PROGRAM P_IncAusstossV
VAR
END_VAR

IF DB6.rAusstossverz < 0.91 THEN
	DB6.rAusstossverz := DB6.rAusstossverz + 0.1;
	DB6.nAusstossverz := REAL_TO_INT(DB6.rAusstossverz * 1000);
END_IF

END_PROGRAM

(* stored: Version 1.1.0.1, ProductVersion 3.1.4024.3
   POU P_IncAusstossV: Id {639d29f2-d485-42df-b344-09290d0fd139}, SpecialFunc None *)
